// TIA Portal project "Nastro_26_01_2021" (V16)

(* hardware
DEVICE "S7-1200 station_1"  S7-1200 Station
   slot 0: "Rack_0"  S7-1200 Rack  Rack  V1.0
   slot 1: "PLC_1"  CPU 1215C DC/DC/Rly  6ES7 215-1HG40-0XB0  V4.4
*)

// ===== PLC "PLC_1"  CPU 1215C DC/DC/Rly =====

VAR_GLOBAL   // PLC tag table "Tabella_Dati_standard"
   "BC_inizio" AT %I0.0 : Bool;
   "BC_fine" AT %I0.1 : Bool;
   "Avanti_Nastro" AT %Q0.0 : Bool;
   "Indietro_Nastro" AT %Q0.1 : Bool;
   "Passi_0" AT %M0.0 : Bool;
   "Passo_1" AT %M0.1 : Bool;
   "Passo_2" AT %M0.2 : Bool;
   "Passo_3" AT %M0.3 : Bool;
   "M_timer" AT %M1.0 : Bool;
   "M_cicli" AT %M1.1 : Bool;
END_VAR

DATA_BLOCK "Blocco_Dati_HMI"   // DB1
{ S7_Optimized_Access := 'TRUE' }
VERSION : 0.1
   VAR
      jog_ripristino : Bool;
      jog_start : Bool;
   END_VAR
BEGIN
END_DATA_BLOCK

// folder: System blocks/Program resources

DATA_BLOCK "IEC_Timer_0_DB"   // DB2
{ S7_Optimized_Access := 'TRUE' }
AUTHOR : Simatic
FAMILY : IEC
NAME : IEC_TMR
VERSION : 1.0
// stored: InstanceOfName IEC_TIMER
"IEC_TIMER"
BEGIN
END_DATA_BLOCK

DATA_BLOCK "Tempo di Lavorazione"   // DB3
{ S7_Optimized_Access := 'TRUE' }
AUTHOR : Simatic
FAMILY : IEC
NAME : IEC_TMR
VERSION : 1.0
// stored: InstanceOfName IEC_TIMER
"IEC_TIMER"
BEGIN
END_DATA_BLOCK

DATA_BLOCK "Numero_Cicli"   // DB4
{ S7_Optimized_Access := 'TRUE' }
AUTHOR : Simatic
FAMILY : IEC
NAME : CNTR
VERSION : 1.0
// stored: InstanceOfName IEC_COUNTER
"IEC_COUNTER"
BEGIN
END_DATA_BLOCK

DATA_BLOCK "Conta_Cicli"   // DB5
{ S7_Optimized_Access := 'TRUE' }
AUTHOR : Simatic
FAMILY : IEC
NAME : CNTR
VERSION : 1.0
// stored: InstanceOfName IEC_COUNTER
"IEC_COUNTER"
BEGIN
END_DATA_BLOCK

// folder: (top level)

FUNCTION "Ripristino" : Void   // FC1, LAD
{ S7_Optimized_Access := 'TRUE' }
VERSION : 0.1
BEGIN

REGION Network 1
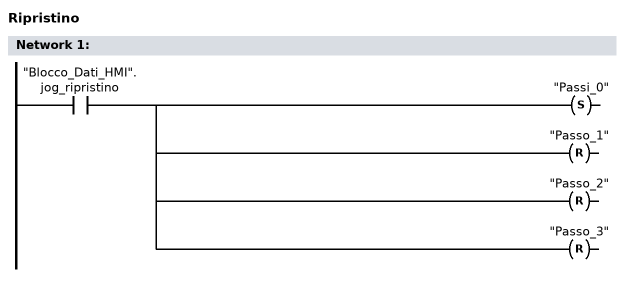
   RUNG wire#powerrail
      Contact( "Blocco_Dati_HMI".jog_ripristino )
      wire#w1
      S_Coil( "Passi_0" )
   END_RUNG
   RUNG wire#w1
      R_Coil( "Passo_1" )
   END_RUNG
   RUNG wire#w1
      R_Coil( "Passo_2" )
   END_RUNG
   RUNG wire#w1
      R_Coil( "Passo_3" )
   END_RUNG
   // the same network as SCL:
   IF "Blocco_Dati_HMI".jog_ripristino THEN
       "Passi_0" := TRUE;
       "Passo_1" := FALSE;
       "Passo_2" := FALSE;
       "Passo_3" := FALSE;
   END_IF;
END_REGION
END_FUNCTION

FUNCTION "Struttura_dei_Passi" : Void   // FC2, LAD
{ S7_Optimized_Access := 'TRUE' }
VERSION : 0.1
   VAR_TEMP   // added for the SCL form of the ladder/FBD networks
      _w1 : Bool;
   END_VAR
BEGIN

REGION Network 1
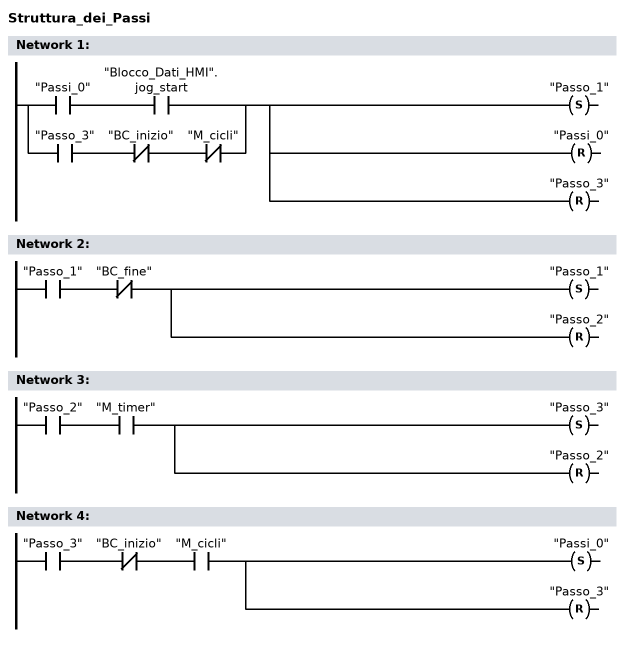
   RUNG wire#powerrail
      Contact( "Passi_0" )
      Contact( "Blocco_Dati_HMI".jog_start )
      wire#w1
      S_Coil( "Passo_1" )
   END_RUNG
   RUNG wire#powerrail
      Contact( "Passo_3" )
      I_Contact( "BC_inizio" )
      I_Contact( "M_cicli" )
   END_RUNG wire#w1
   RUNG wire#w1
      R_Coil( "Passi_0" )
   END_RUNG
   RUNG wire#w1
      R_Coil( "Passo_3" )
   END_RUNG
   // the same network as SCL:
   IF ("Passi_0" AND "Blocco_Dati_HMI".jog_start) OR ("Passo_3" AND NOT "BC_inizio" AND NOT "M_cicli") THEN
       "Passo_1" := TRUE;
   END_IF;
   #_w1 := ("Passi_0" AND "Blocco_Dati_HMI".jog_start) OR ("Passo_3" AND NOT "BC_inizio" AND NOT "M_cicli");
   IF #_w1 THEN
       "Passi_0" := FALSE;
       "Passo_3" := FALSE;
   END_IF;
END_REGION

REGION Network 2
   RUNG wire#powerrail
      Contact( "Passo_1" )
      I_Contact( "BC_fine" )
      wire#w1
      S_Coil( "Passo_1" )
   END_RUNG
   RUNG wire#w1
      R_Coil( "Passo_2" )
   END_RUNG
   // the same network as SCL:
   #_w1 := "Passo_1" AND NOT "BC_fine";
   IF #_w1 THEN
       "Passo_1" := TRUE;
       "Passo_2" := FALSE;
   END_IF;
END_REGION

REGION Network 3
   RUNG wire#powerrail
      Contact( "Passo_2" )
      Contact( "M_timer" )
      wire#w1
      S_Coil( "Passo_3" )
   END_RUNG
   RUNG wire#w1
      R_Coil( "Passo_2" )
   END_RUNG
   // the same network as SCL:
   IF "Passo_2" AND "M_timer" THEN
       "Passo_3" := TRUE;
       "Passo_2" := FALSE;
   END_IF;
END_REGION

REGION Network 4
   RUNG wire#powerrail
      Contact( "Passo_3" )
      I_Contact( "BC_inizio" )
      Contact( "M_cicli" )
      wire#w1
      S_Coil( "Passi_0" )
   END_RUNG
   RUNG wire#w1
      R_Coil( "Passo_3" )
   END_RUNG
   // the same network as SCL:
   IF "Passo_3" AND NOT "BC_inizio" AND "M_cicli" THEN
       "Passi_0" := TRUE;
       "Passo_3" := FALSE;
   END_IF;
END_REGION
END_FUNCTION

FUNCTION "Attivazione_delle_Uscite" : Void   // FC3, LAD
{ S7_Optimized_Access := 'TRUE' }
VERSION : 0.1
BEGIN

REGION Network 1
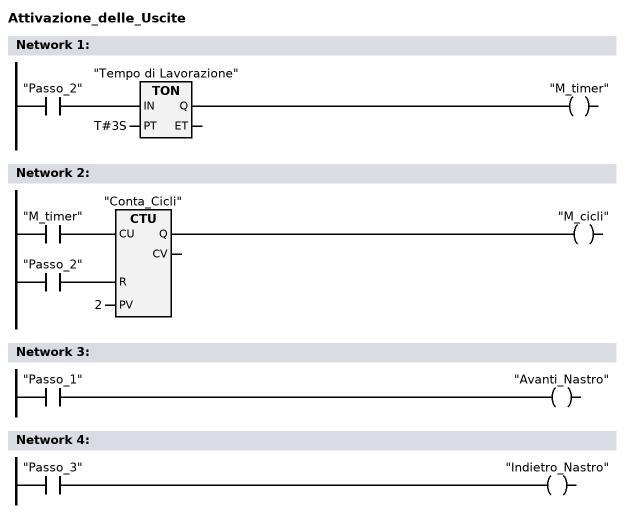
   "Tempo di Lavorazione".TON(IN := "Passo_2", PT := T#3S);
   "M_timer" := "Tempo di Lavorazione".Q;
END_REGION

REGION Network 2
   "Conta_Cicli".CTU(CU := "M_timer", R := "Passo_2", PV := 2);
   "M_cicli" := "Conta_Cicli".Q;
END_REGION

REGION Network 3
   RUNG wire#powerrail
      Contact( "Passo_1" )
      Coil( "Avanti_Nastro" )
   END_RUNG
   // the same network as SCL:
   "Avanti_Nastro" := "Passo_1";
END_REGION

REGION Network 4
   RUNG wire#powerrail
      Contact( "Passo_3" )
      Coil( "Indietro_Nastro" )
   END_RUNG
   // the same network as SCL:
   "Indietro_Nastro" := "Passo_3";
END_REGION
END_FUNCTION

ORGANIZATION_BLOCK "Main"   // OB1, LAD, ProgramCycle
TITLE = "Main Program Sweep (Cycle)"
{ S7_Optimized_Access := 'TRUE' }
VERSION : 0.1
   VAR_INPUT
      Initial_Call : Bool;   // Initial call of this OB
      Remanence : Bool;   // =True, if remanent data are available
   END_VAR
BEGIN
END_ORGANIZATION_BLOCK